Universal Robots PolyScope program: 12.urp

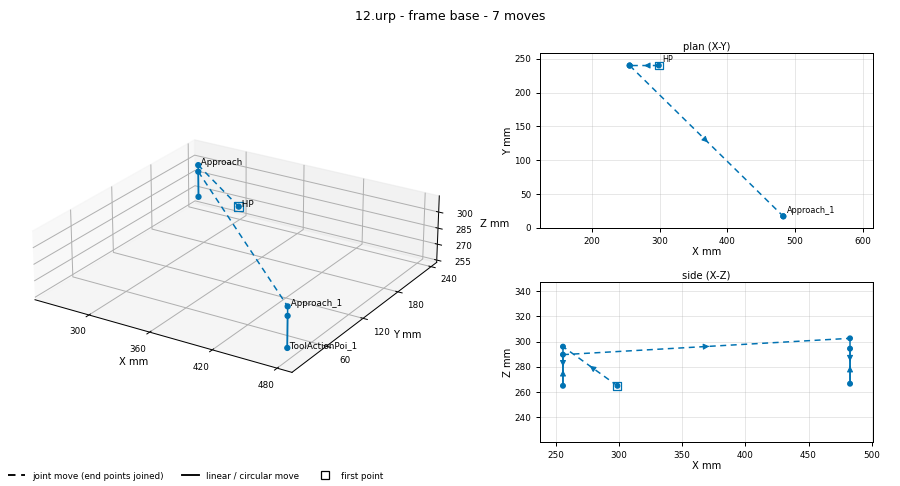
[picture p0: tool path of 12.urp in frame base, 7 of 7 moves have a stored position in this frame; points joined in program order, loops and branches not executed]
Program 12 (installation=default directory=/programs/Students createdIn=5.11.9.1010452 lastSavedIn=5.11.9.1010452 robotSerialNumber=20225200364)
Calibrated DH parameters: a=[0.00002, -0.569483, -0.54992, -0.00001, -0.000036, 0]; d=[0.180894, -146.691669, 192.918669, -46.053088, 0.119778, 0.115602]; alpha=[1.571425, -0.001534, 0.003359, 1.568739, -1.571477, 0]; deltaTheta=[0, 0.376258, -0.101074, -0.275185, -0.000002, 0]
Robot Program (runOnlyOnce=false)
  URCap RG Grip (OnRobot, OnRobot A/S) dataModel(rg-target-force=40.0, workpiece-lost=true, Variable(key=on_return, variable(name=on_return)))
  MoveJ speed 60 deg/s, acceleration 80 deg/s^2 (useActiveTCP=true) feature=Base
    Waypoint HP: TCP in base x=298.742 y=239.99 z=265.066 mm, rx=2.2309 ry=-2.1851 rz=-0.032 rad; joints [65.347, -96.187, -129.782, -224.671, -91.62, -115.552] deg
  Loop Counting (count=3) loopVariable(name=Loop_1)
    URCap Palletizing (polyscope-pallet-impl, Universal Robots) dataModel(palletFeature=Base, isPalletizing=true, Length(key=objectHeight value=0.00001 unit=M), Variable(key=name, variable(name=Pallet_1)), Variable(key=globalCountingVariable, variable(name=Pallet_1_cnt_1, initializeExpression=1)), Variable(key=layerNumberVariable, variable(name=Pallet_1_lno, initializeExpression=1)), Variable(key=layerCountingVariable, variable(name=Pallet_1_lct, initializeExpression=1)), Variable(key=handleSeparatorVariable, variable(name=Pallet_1_sep, initializeExpression=False)), Variable(key=totalCountVariable, variable(name=Pallet_1_tct, initializeExpression=1)), Variable(key=referencePoint, variable(featureName=referencePoint)), Variable(key=separatorPoint, variable(featureName=separatorPoint))); state(isChildrenLocked=true)
      URCap Patterns (polyscope-pallet-impl, Universal Robots) state(isChildrenLocked=true)
        URCap Pattern (polyscope-pallet-impl, Universal Robots) dataModel(UUID=4db255ee-a530-4199-8934-97ba4d854a09, patternType=LINE, objects=3, Variable(key=nameVariable, variable(name=Line_Pattern_1))); state(isChildrenLocked=true)
          URCap Item (polyscope-pallet-impl, Universal Robots) dataModel(UUID=7e993e0f-8f50-41e7-b3c8-4f6520dbf927, patternType=LINE, index=0, calibrationDeltaTheta=[-2.1094217540068572E-7, 0.37625772532806073, -0.10107441100396769, -0.2751850025766889, -1.8024952768980196E-6, 2.9402326063437956E-8], calibrationA=[2.0416891277915125E-5, -0.5694828868469309, -0.5499202125525207, -9.504674691390763E-6, -3.603723657207661E-5, 0.0], calibrationD=[0.1808937726775539, -146.69166934821124, 192.91866861971778, -46.05308757405963, 0.11977780403821288, 0.11560212559305974], calibrationAlpha=[1.5714252480212174, -0.0015337665762078037, 0.0033588312559612306, 1.5687392298942362, -1.5714772428732047, 0.0], calibrationJointChecksum=[-1490546360, -1456574554, -1506622700, -1493399207, -1492840923, -1492940558], calibrationStatus=2, calibrationValidChecksum=true, baseToFeature=[0.0, 0.0, 0.0, 0.0, 0.0, 0.0], TCPOffset=[2.3631021561498766E-6, 7.198250485340729E-6, 1.244139811595879E-5, -3.576711212253427E-5, 5.463755960822963E-5, 2.2123390688281095E-5], Variable(key=variable, variable(name=StartItem_1)), JointPositions(key=jointpositions, JointPosition(key=[1], Angle(key=pos value=1.264006 unit=RAD)), JointPosition(key=[2], Angle(key=pos value=-1.6221 unit=RAD)), JointPosition(key=[3], Angle(key=pos value=-2.327859 unit=RAD)), JointPosition(key=[4], Angle(key=pos value=-3.912183 unit=RAD)), JointPosition(key=[5], Angle(key=pos value=-1.601024 unit=RAD)), JointPosition(key=[6], Angle(key=pos value=-1.893251 unit=RAD))))
          URCap Item (polyscope-pallet-impl, Universal Robots) dataModel(UUID=744d39a8-2258-49f5-9eba-0e5eedd8a8bf, patternType=LINE, index=1, calibrationDeltaTheta=[-2.1094217540068572E-7, 0.37625772532806073, -0.10107441100396769, -0.2751850025766889, -1.8024952768980196E-6, 2.9402326063437956E-8], calibrationA=[2.0416891277915125E-5, -0.5694828868469309, -0.5499202125525207, -9.504674691390763E-6, -3.603723657207661E-5, 0.0], calibrationD=[0.1808937726775539, -146.69166934821124, 192.91866861971778, -46.05308757405963, 0.11977780403821288, 0.11560212559305974], calibrationAlpha=[1.5714252480212174, -0.0015337665762078037, 0.0033588312559612306, 1.5687392298942362, -1.5714772428732047, 0.0], calibrationJointChecksum=[-1490546360, -1456574554, -1506622700, -1493399207, -1492840923, -1492940558], calibrationStatus=2, calibrationValidChecksum=true, baseToFeature=[0.0, 0.0, 0.0, 0.0, 0.0, 0.0], TCPOffset=[-2.2334165447751575E-5, -1.0734787209143448E-7, -2.1984189987944713E-5, 2.4451271934751318E-5, -6.0457600479340426E-5, 1.8015936155033457E-5], Variable(key=variable, variable(name=EndItem_1)), JointPositions(key=jointpositions, JointPosition(key=[1], Angle(key=pos value=1.264006 unit=RAD)), JointPosition(key=[2], Angle(key=pos value=-1.6221 unit=RAD)), JointPosition(key=[3], Angle(key=pos value=-2.327859 unit=RAD)), JointPosition(key=[4], Angle(key=pos value=-3.912183 unit=RAD)), JointPosition(key=[5], Angle(key=pos value=-1.601024 unit=RAD)), JointPosition(key=[6], Angle(key=pos value=-1.893251 unit=RAD))))
      URCap Layers (polyscope-pallet-impl, Universal Robots) dataModel(separators=[false], selectedPatterns=[4db255ee-a530-4199-8934-97ba4d854a09])
      URCap At Each Item (polyscope-pallet-impl, Universal Robots) dataModel(selectedPattern=4db255ee-a530-4199-8934-97ba4d854a09, selectedPosition=7e993e0f-8f50-41e7-b3c8-4f6520dbf927, Approach_calibrationDeltaTheta=[-2.1094217540068572E-7, 0.37625772532806073, -0.10107441100396769, -0.2751850025766889, -1.8024952768980196E-6, 2.9402326063437956E-8], Approach_calibrationA=[2.0416891277915125E-5, -0.5694828868469309, -0.5499202125525207, -9.504674691390763E-6, -3.603723657207661E-5, 0.0], Approach_calibrationD=[0.1808937726775539, -146.69166934821124, 192.91866861971778, -46.05308757405963, 0.11977780403821288, 0.11560212559305974], Approach_calibrationAlpha=[1.5714252480212174, -0.0015337665762078037, 0.0033588312559612306, 1.5687392298942362, -1.5714772428732047, 0.0], Approach_calibrationJointChecksum=[-1490546360, -1456574554, -1506622700, -1493399207, -1492840923, -1492940558], Approach_calibrationStatus=2, Approach_calibrationValidChecksum=true, Approach_baseToFeature=[0.0, 0.0, 0.0, 0.0, 0.0, 0.0], Approach_TCPOffset=[3.3548432041563547E-6, -4.1201008819102825E-6, -1.2111014214444271E-5, 3.1354525010668334E-5, -1.5228688827521043E-6, 2.6578353226408743E-5], Exit_calibrationDeltaTheta=[-2.1094217540068572E-7, 0.37625772532806073, -0.10107441100396769, -0.2751850025766889, -1.8024952768980196E-6, 2.9402326063437956E-8], Exit_calibrationA=[2.0416891277915125E-5, -0.5694828868469309, -0.5499202125525207, -9.504674691390763E-6, -3.603723657207661E-5, 0.0], Exit_calibrationD=[0.1808937726775539, -146.69166934821124, 192.91866861971778, -46.05308757405963, 0.11977780403821288, 0.11560212559305974], Exit_calibrationAlpha=[1.5714252480212174, -0.0015337665762078037, 0.0033588312559612306, 1.5687392298942362, -1.5714772428732047, 0.0], Exit_calibrationJointChecksum=[-1490546360, -1456574554, -1506622700, -1493399207, -1492840923, -1492940558], Exit_calibrationStatus=2, Exit_calibrationValidChecksum=true, Exit_baseToFeature=[0.0, 0.0, 0.0, 0.0, 0.0, 0.0], Exit_TCPOffset=[1.7494479089802395E-5, 1.6305084660217517E-6, -8.35008940519577E-6, 1.8517313618601004E-5, -7.774464705213298E-5, 1.9657845672314753E-5], currentWizardState=LANDING, Pose(key=refBaseToFeature, Position(key=posePosition, Length(key=X value=0 unit=M), Length(key=Y value=0 unit=M), Length(key=Z value=0 unit=M)), Rotation(key=poseRotation, Angle(key=RX value=0 unit=RAD), Angle(key=RY value=0 unit=RAD), Angle(key=RZ value=0 unit=RAD))), Pose(key=refPose, Position(key=posePosition, Length(key=X value=0.255641 unit=M), Length(key=Y value=0.239981 unit=M), Length(key=Z value=0.265075 unit=M)), Rotation(key=poseRotation, Angle(key=RX value=2.230448 unit=RAD), Angle(key=RY value=-2.184713 unit=RAD), Angle(key=RZ value=-0.032849 unit=RAD))), JointPositions(key=Approach_jointpositions, JointPosition(key=[1], Angle(key=pos value=1.263923 unit=RAD)), JointPosition(key=[2], Angle(key=pos value=-1.574285 unit=RAD)), JointPosition(key=[3], Angle(key=pos value=-2.302059 unit=RAD)), JointPosition(key=[4], Angle(key=pos value=-3.98587 unit=RAD)), JointPosition(key=[5], Angle(key=pos value=-1.601224 unit=RAD)), JointPosition(key=[6], Angle(key=pos value=-1.893558 unit=RAD))), JointPositions(key=Exit_jointpositions, JointPosition(key=[1], Angle(key=pos value=1.263944 unit=RAD)), JointPosition(key=[2], Angle(key=pos value=-1.583694 unit=RAD)), JointPosition(key=[3], Angle(key=pos value=-2.307598 unit=RAD)), JointPosition(key=[4], Angle(key=pos value=-3.970921 unit=RAD)), JointPosition(key=[5], Angle(key=pos value=-1.601189 unit=RAD)), JointPosition(key=[6], Angle(key=pos value=-1.893487 unit=RAD))))
        URCap Generated Movements (polyscope-pallet-impl, Universal Robots) state(isChildrenLocked=true)
          MoveJ speed 60 deg/s, acceleration 80 deg/s^2 (useActiveTCP=true) feature=referencePoint
            Waypoint Approach: TCP in base x=255.646 y=239.978 z=296.089 mm, rx=2.2304 ry=-2.1848 rz=-0.0328 rad; joints [72.417, -90.199, -131.898, -228.375, -91.742, -108.492] deg; TCP offset x=0 y=0 z=0 mm, rx=0 ry=0 rz=0 rad; feature pose in base x=255.641 y=239.981 z=265.075 mm, rx=2.2304 ry=-2.1847 rz=-0.0328 rad
          MoveL speed 250 mm/s, acceleration 1200 mm/s^2 (useActiveTCP=true) feature(featureName=referencePoint)
            Waypoint ToolActionPoint: TCP in base x=255.641 y=239.981 z=265.075 mm, rx=2.2304 ry=-2.1847 rz=-0.0328 rad; joints [72.423, -92.941, -133.377, -224.152, -91.733, -108.473] deg; TCP offset x=0 y=0 z=0 mm, rx=0 ry=0 rz=0 rad
          Folder Tool action
            URCap RG Grip (OnRobot, OnRobot A/S) dataModel(rg-target-force=40.0)
          MoveL speed 250 mm/s, acceleration 1200 mm/s^2 (useActiveTCP=true) feature(featureName=referencePoint)
            Waypoint Exit_1: TCP in base x=255.64 y=239.964 z=289.737 mm, rx=2.2305 ry=-2.1848 rz=-0.0329 rad; joints [72.418, -90.735, -132.217, -227.515, -91.742, -108.489] deg; TCP offset x=0 y=0 z=0 mm, rx=0 ry=0 rz=0 rad
    URCap Palletizing (polyscope-pallet-impl, Universal Robots) dataModel(palletFeature=Base, isPalletizing=true, Variable(key=name, variable(name=Pallet_2)), Variable(key=globalCountingVariable, variable(name=Pallet_2_cnt, initializeExpression=1)), Variable(key=layerNumberVariable, variable(name=Pallet_2_lno, initializeExpression=1)), Variable(key=layerCountingVariable, variable(name=Pallet_2_lct, initializeExpression=1)), Variable(key=handleSeparatorVariable, variable(name=Pallet_2_sep, initializeExpression=False)), Variable(key=totalCountVariable, variable(name=Pallet_2_tct, initializeExpression=1)), Variable(key=referencePoint, variable(featureName=referencePoin_1)), Variable(key=separatorPoint, variable(featureName=separatorPoin_1)), Length(key=objectHeight value=0.00001 unit=M)); state(isChildrenLocked=true)
      URCap Patterns (polyscope-pallet-impl, Universal Robots) state(isChildrenLocked=true)
        URCap Pattern (polyscope-pallet-impl, Universal Robots) dataModel(UUID=90cc6f69-a1d3-4d9f-b98e-0ae263274573, patternType=LINE, objects=3, Variable(key=nameVariable, variable(name=Line_Pattern_2))); state(isChildrenLocked=true)
          URCap Item (polyscope-pallet-impl, Universal Robots) dataModel(UUID=3c1ecc6b-1ec8-44b8-9fad-3ff7e7664849, patternType=LINE, index=0, calibrationDeltaTheta=[-2.1094217540068572E-7, 0.37625772532806073, -0.10107441100396769, -0.2751850025766889, -1.8024952768980196E-6, 2.9402326063437956E-8], calibrationA=[2.0416891277915125E-5, -0.5694828868469309, -0.5499202125525207, -9.504674691390763E-6, -3.603723657207661E-5, 0.0], calibrationD=[0.1808937726775539, -146.69166934821124, 192.91866861971778, -46.05308757405963, 0.11977780403821288, 0.11560212559305974], calibrationAlpha=[1.5714252480212174, -0.0015337665762078037, 0.0033588312559612306, 1.5687392298942362, -1.5714772428732047, 0.0], calibrationJointChecksum=[-1490546360, -1456574554, -1506622700, -1493399207, -1492840923, -1492940558], calibrationStatus=2, calibrationValidChecksum=true, baseToFeature=[0.0, 0.0, 0.0, 0.0, 0.0, 0.0], TCPOffset=[-9.44477072217266E-6, -2.084231430998784E-6, 4.473857629028188E-6, 3.8873744161357277E-5, -3.490594776559334E-5, -2.321802329315874E-5], Variable(key=variable, variable(name=StartItem_2)), JointPositions(key=jointpositions, JointPosition(key=[1], Angle(key=pos value=0.401031 unit=RAD)), JointPosition(key=[2], Angle(key=pos value=-1.83355 unit=RAD)), JointPosition(key=[3], Angle(key=pos value=-2.067749 unit=RAD)), JointPosition(key=[4], Angle(key=pos value=-3.979168 unit=RAD)), JointPosition(key=[5], Angle(key=pos value=-1.585404 unit=RAD)), JointPosition(key=[6], Angle(key=pos value=-2.756364 unit=RAD))))
          URCap Item (polyscope-pallet-impl, Universal Robots) dataModel(UUID=d36ca927-4d46-47bb-abea-4cc36ed8b6d5, patternType=LINE, index=1, calibrationDeltaTheta=[-2.1094217540068572E-7, 0.37625772532806073, -0.10107441100396769, -0.2751850025766889, -1.8024952768980196E-6, 2.9402326063437956E-8], calibrationA=[2.0416891277915125E-5, -0.5694828868469309, -0.5499202125525207, -9.504674691390763E-6, -3.603723657207661E-5, 0.0], calibrationD=[0.1808937726775539, -146.69166934821124, 192.91866861971778, -46.05308757405963, 0.11977780403821288, 0.11560212559305974], calibrationAlpha=[1.5714252480212174, -0.0015337665762078037, 0.0033588312559612306, 1.5687392298942362, -1.5714772428732047, 0.0], calibrationJointChecksum=[-1490546360, -1456574554, -1506622700, -1493399207, -1492840923, -1492940558], calibrationStatus=2, calibrationValidChecksum=true, baseToFeature=[0.0, 0.0, 0.0, 0.0, 0.0, 0.0], TCPOffset=[3.1019666802949847E-6, 2.0266897479914725E-5, 1.795182694624975E-5, -2.2518676562975244E-5, 2.970293730321597E-5, -2.0235678618555696E-5], Variable(key=variable, variable(name=EndItem_2)), JointPositions(key=jointpositions, JointPosition(key=[1], Angle(key=pos value=0.454853 unit=RAD)), JointPosition(key=[2], Angle(key=pos value=-1.761409 unit=RAD)), JointPosition(key=[3], Angle(key=pos value=-2.180395 unit=RAD)), JointPosition(key=[4], Angle(key=pos value=-3.937971 unit=RAD)), JointPosition(key=[5], Angle(key=pos value=-1.586822 unit=RAD)), JointPosition(key=[6], Angle(key=pos value=-2.702453 unit=RAD))))
      URCap Layers (polyscope-pallet-impl, Universal Robots) dataModel(separators=[false], selectedPatterns=[90cc6f69-a1d3-4d9f-b98e-0ae263274573])
      URCap At Each Item (polyscope-pallet-impl, Universal Robots) dataModel(selectedPattern=90cc6f69-a1d3-4d9f-b98e-0ae263274573, selectedPosition=3c1ecc6b-1ec8-44b8-9fad-3ff7e7664849, Approach_calibrationDeltaTheta=[-2.1094217540068572E-7, 0.37625772532806073, -0.10107441100396769, -0.2751850025766889, -1.8024952768980196E-6, 2.9402326063437956E-8], Approach_calibrationA=[2.0416891277915125E-5, -0.5694828868469309, -0.5499202125525207, -9.504674691390763E-6, -3.603723657207661E-5, 0.0], Approach_calibrationD=[0.1808937726775539, -146.69166934821124, 192.91866861971778, -46.05308757405963, 0.11977780403821288, 0.11560212559305974], Approach_calibrationAlpha=[1.5714252480212174, -0.0015337665762078037, 0.0033588312559612306, 1.5687392298942362, -1.5714772428732047, 0.0], Approach_calibrationJointChecksum=[-1490546360, -1456574554, -1506622700, -1493399207, -1492840923, -1492940558], Approach_calibrationStatus=2, Approach_calibrationValidChecksum=true, Approach_baseToFeature=[0.0, 0.0, 0.0, 0.0, 0.0, 0.0], Approach_TCPOffset=[3.0045348046669855E-5, 2.5858295621739025E-5, -4.239767628810842E-6, -3.602691844660108E-5, 9.287178040097534E-7, 3.287105858955803E-5], Exit_calibrationDeltaTheta=[-2.1094217540068572E-7, 0.37625772532806073, -0.10107441100396769, -0.2751850025766889, -1.8024952768980196E-6, 2.9402326063437956E-8], Exit_calibrationA=[2.0416891277915125E-5, -0.5694828868469309, -0.5499202125525207, -9.504674691390763E-6, -3.603723657207661E-5, 0.0], Exit_calibrationD=[0.1808937726775539, -146.69166934821124, 192.91866861971778, -46.05308757405963, 0.11977780403821288, 0.11560212559305974], Exit_calibrationAlpha=[1.5714252480212174, -0.0015337665762078037, 0.0033588312559612306, 1.5687392298942362, -1.5714772428732047, 0.0], Exit_calibrationJointChecksum=[-1490546360, -1456574554, -1506622700, -1493399207, -1492840923, -1492940558], Exit_calibrationStatus=2, Exit_calibrationValidChecksum=true, Exit_baseToFeature=[0.0, 0.0, 0.0, 0.0, 0.0, 0.0], Exit_TCPOffset=[-1.0708969732610082E-5, 6.231826172042876E-6, -9.708850538192593E-6, 7.141189650678229E-6, -3.9146305404301506E-5, -1.6725715901147367E-5], currentWizardState=LANDING, Pose(key=refBaseToFeature, Position(key=posePosition, Length(key=X value=0 unit=M), Length(key=Y value=0 unit=M), Length(key=Z value=0 unit=M)), Rotation(key=poseRotation, Angle(key=RX value=0 unit=RAD), Angle(key=RY value=0 unit=RAD), Angle(key=RZ value=0 unit=RAD))), Pose(key=refPose, Position(key=posePosition, Length(key=X value=0.482843 unit=M), Length(key=Y value=0.01703 unit=M), Length(key=Z value=0.266713 unit=M)), Rotation(key=poseRotation, Angle(key=RX value=2.23051 unit=RAD), Angle(key=RY value=-2.184725 unit=RAD), Angle(key=RZ value=-0.032847 unit=RAD))), JointPositions(key=Approach_jointpositions, JointPosition(key=[1], Angle(key=pos value=0.400998 unit=RAD)), JointPosition(key=[2], Angle(key=pos value=-1.789656 unit=RAD)), JointPosition(key=[3], Angle(key=pos value=-2.042655 unit=RAD)), JointPosition(key=[4], Angle(key=pos value=-4.04811 unit=RAD)), JointPosition(key=[5], Angle(key=pos value=-1.585582 unit=RAD)), JointPosition(key=[6], Angle(key=pos value=-2.756641 unit=RAD))), JointPositions(key=Exit_jointpositions, JointPosition(key=[1], Angle(key=pos value=0.401009 unit=RAD)), JointPosition(key=[2], Angle(key=pos value=-1.79927 unit=RAD)), JointPosition(key=[3], Angle(key=pos value=-2.048691 unit=RAD)), JointPosition(key=[4], Angle(key=pos value=-4.032459 unit=RAD)), JointPosition(key=[5], Angle(key=pos value=-1.585548 unit=RAD)), JointPosition(key=[6], Angle(key=pos value=-2.756579 unit=RAD))))
        URCap Generated Movements (polyscope-pallet-impl, Universal Robots) state(isChildrenLocked=true)
          MoveJ speed 60 deg/s, acceleration 80 deg/s^2 (useActiveTCP=true) feature=referencePoin_1
            Waypoint Approach_1: TCP in base x=482.818 y=17 z=302.651 mm, rx=2.2305 ry=-2.1847 rz=-0.0329 rad; joints [22.973, -102.538, -117.038, -231.941, -90.848, -157.945] deg; TCP offset x=0 y=0 z=0 mm, rx=0 ry=0 rz=0 rad; feature pose in base x=482.843 y=17.03 z=266.713 mm, rx=2.2305 ry=-2.1847 rz=-0.0328 rad
          MoveL speed 250 mm/s, acceleration 1200 mm/s^2 (useActiveTCP=true) feature(featureName=referencePoin_1)
            Waypoint ToolActionPoi_1: TCP in base x=482.843 y=17.03 z=266.713 mm, rx=2.2305 ry=-2.1847 rz=-0.0328 rad; joints [22.978, -105.054, -118.474, -227.987, -90.838, -157.929] deg; TCP offset x=0 y=0 z=0 mm, rx=0 ry=0 rz=0 rad
          Folder Tool action
            URCap RG Grip (OnRobot, OnRobot A/S) dataModel(rg-target-force=40.0)
          MoveL speed 250 mm/s, acceleration 1200 mm/s^2 (useActiveTCP=true) feature(featureName=referencePoin_1)
            Waypoint Exit_2: TCP in base x=482.837 y=17.041 z=294.496 mm, rx=2.2306 ry=-2.1847 rz=-0.0329 rad; joints [22.977, -103.089, -117.382, -231.043, -90.847, -157.94] deg; TCP offset x=0 y=0 z=0 mm, rx=0 ry=0 rz=0 rad
